FUNCTION_BLOCK PositionMarkerFS (* Moves a VT marker object to reflect an incoming REAL value — accepts PositionMarker_S struct, clamps to the marker's travel range, drives Q_ChildPosition *)
  (* Standard: ISO 11783-6; Description: Copyright (c) 2026 Meisterschulen am Ostbahnhof This program and the accompanying materials are made available under the terms of the Eclipse Public License 2.0 which is available at https://www.eclipse.org/legal/epl-2.0/ SPDX-License-Identifier: EPL-2.0 Wraps a single Q_ChildPosition instance (ISO 11783-6 F.16) that moves a marker object (e.g. a triangle) within its container, given an arbitrary REAL value (from any source - a VT InputNumber via NumericValue_PHYS, a sensor, or anything else). stObj is snapshotted once at INIT via F_MOVE, matching the ScrollFS/Q_NumericValue_PHYS pattern. The incoming value is offset by stObj.r32Center, clamped to stObj.r32MinPos..r32MaxPos (reporting xOver/xUnder), then integerized once for Q_ChildPosition.s16Xposition. s16Yposition is a fixed passthrough of stObj.s16YPosition. *)
  (* Version 1.1, 2026-09-05, Franz Höpfinger, Meisterschulen am Ostbahnhof, Add xScale flag, passed through to the internal MoveMarker (Q_ChildPosition) *)
  (* Version 1.0, 2026-09-05, Franz Höpfinger, Meisterschulen am Ostbahnhof, initial API and implementation and/or initial documentation *)
  PACKAGE isobus::UT::Q;
  IMPORT isobus::utils::childposition::PositionMarker_S;
  IMPORT isobus::UT::Q::Q_ChildPosition;
  IMPORT iec61131::selection::F_MOVE;
  IMPORT iec61131::arithmetic::F_ADD;
  IMPORT iec61131::conversion::F_REAL_TO_INT;
  IMPORT logiBUS::signalprocessing::clamp::F_ClampReal;
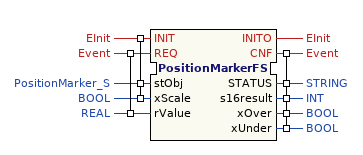
  EVENT_INPUT
    INIT : EInit WITH stObj, xScale; (* Service Initialization *)
    REQ WITH rValue; (* Move the marker to reflect a new value *)
  END_EVENT
  EVENT_OUTPUT
    INITO : EInit; (* Initialization Confirm *)
    CNF WITH STATUS, s16result, xOver, xUnder; (* Confirmation of Requested Service *)
  END_EVENT
  VAR_INPUT
    stObj : isobus::utils::childposition::PositionMarker_S; (* Marker object pool properties (child/parent IDs, travel bounds, center offset), snapshotted at INIT *)
    xScale : BOOL := FALSE; (* FALSE (default) = bypass, send s16Xposition/s16Yposition through unchanged. TRUE = scale them by the DM/SKM factor for stObj.u16ParentId. Passed straight through to the internal MoveMarker (Q_ChildPosition). *)
    rValue : REAL; (* Physical value to display - from any source, not limited to NumericValue_PHYS *)
  END_VAR
  VAR_OUTPUT
    STATUS : STRING; (* Service Status - passthrough from the internal Q_ChildPosition *)
    s16result : INT; (* retval - passthrough from the internal Q_ChildPosition, see Q_ChildPosition *)
    xOver : BOOL; (* rValue (after adding stObj.r32Center) exceeded stObj.r32MaxPos and was clamped *)
    xUnder : BOOL; (* rValue (after adding stObj.r32Center) fell below stObj.r32MinPos and was clamped *)
  END_VAR
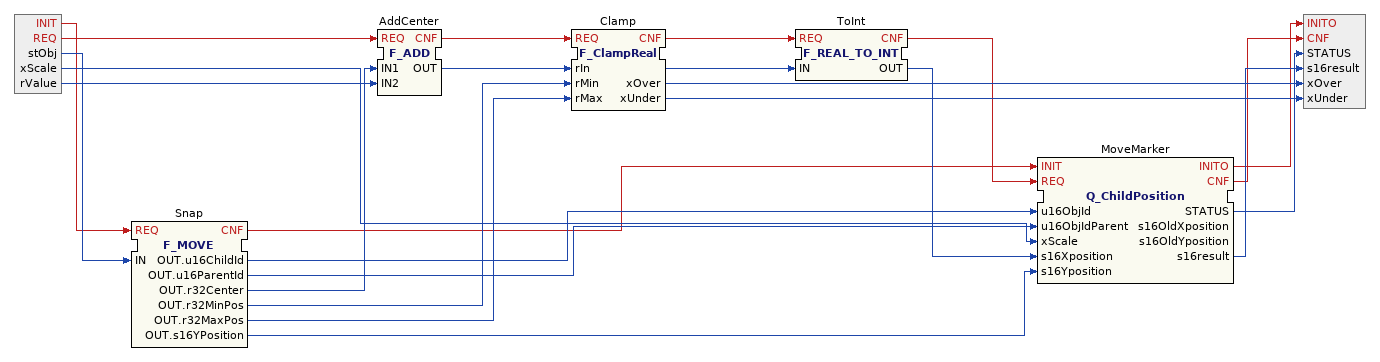
  FBS
    Snap : iec61131::selection::F_MOVE; {SET_ATTRIBUTE(DataType, isobus::utils::childposition::PositionMarker_S)}
    AddCenter : iec61131::arithmetic::F_ADD;
    Clamp : logiBUS::signalprocessing::clamp::F_ClampReal;
    ToInt : iec61131::conversion::F_REAL_TO_INT;
    MoveMarker : isobus::UT::Q::Q_ChildPosition;
  END_FBS
  EVENT_CONNECTIONS
    INIT TO Snap.REQ;
    Snap.CNF TO MoveMarker.INIT;
    REQ TO AddCenter.REQ;
    AddCenter.CNF TO Clamp.REQ;
    Clamp.CNF TO ToInt.REQ;
    ToInt.CNF TO MoveMarker.REQ;
    MoveMarker.INITO TO INITO;
    MoveMarker.CNF TO CNF;
  END_CONNECTIONS
  DATA_CONNECTIONS
    stObj TO Snap.IN;
    Snap.OUT.u16ChildId TO MoveMarker.u16ObjId;
    Snap.OUT.u16ParentId TO MoveMarker.u16ObjIdParent;
    xScale TO MoveMarker.xScale;
    rValue TO AddCenter.IN1;
    Snap.OUT.r32Center TO AddCenter.IN2;
    AddCenter.OUT TO Clamp.rIn;
    Snap.OUT.r32MinPos TO Clamp.rMin;
    Snap.OUT.r32MaxPos TO Clamp.rMax;
    Clamp. TO ToInt.IN;
    ToInt.OUT TO MoveMarker.s16Xposition;
    Snap.OUT.s16YPosition TO MoveMarker.s16Yposition;
    MoveMarker.STATUS TO STATUS;
    MoveMarker.s16result TO s16result;
    Clamp.xOver TO xOver;
    Clamp.xUnder TO xUnder;
  END_CONNECTIONS
END_FUNCTION_BLOCK
